{attribute 'qualified_only'}
VAR_GLOBAL CONSTANT
	nModuleNumber  : UINT := 16;
	NumberOfMovers : INT := 10;
	NumberOfStations : INT := 6;
	TrackLength : LREAL := 4000.0;
	TrackHomePosition : LREAL := 800.0;
	Tracks : UDINT := 1;
END_VAR

(* stored: Version 1.1.0.1, ProductVersion 3.1.4024.11
   GVL SystemParameters: Id {a9d78563-e24a-4bd7-bad1-00d0c27c4244}, ParameterList True *)
